Staubli VAL3: aLight1.pgx

public program aLight1(num nValue (dimensions=1))
begin
  aioSet(aLight1,nValue)
end
